(*******************************************************************************
                          protoc-gen-twincat V0.0.0.0                           
                  https://github.com/TcHaxx/protoc-gen-twincat                  
*******************************************************************************)
TYPE ST_Bar :
STRUCT
	name : STRING;
	age : UDINT;
	email : STRING;
END_STRUCT
END_TYPE

(* stored: Version 1.1.0.1
   DUT ST_Bar: Id {560b6726-45eb-4b96-b924-9775c56c70f5} *)
